FUNCTION_BLOCK HTTP_ENDPOINT_SERVER
  {SET_ATTRIBUTE(OpcUa, POINT.STARTPOINT)}
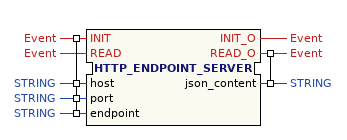
  EVENT_INPUT
    INIT WITH host, port, endpoint;
    READ; {SET_ATTRIBUTE(OpcUa, Method)}
  END_EVENT
  EVENT_OUTPUT
    INIT_O;
    READ_O WITH json_content;
  END_EVENT
  VAR_INPUT
    host : STRING; {SET_ATTRIBUTE(OpcUa, Constant.RUN)}
    port : STRING; {SET_ATTRIBUTE(OpcUa, Constant.RUN)}
    endpoint : STRING; {SET_ATTRIBUTE(OpcUa, Constant.RUN)}
  END_VAR
  VAR_OUTPUT
    json_content : STRING; {SET_ATTRIBUTE(OpcUa, Variable.RUN)}
  END_VAR
END_FUNCTION_BLOCK
